(*
SPDX-FileCopyrightText: © 2026 Oleksandr Tiutyk <trofimich@gmail.com>
SPDX-License-Identifier: MIT
License: https://opensource.org/license/mit
*)

(*!
<summary>Selects whether LogManager supplies no number, a global sequence or a sequence per category.</summary>
<description>
Sequences use counters of requests passing filtering, incremented before the logger call. Numbers represent
attempts rather than successful writes; unsuccessful writes can leave gaps in the output sequence.
</description>
*)
{attribute 'qualified_only'}
{attribute 'strict'}
{attribute 'to_string'}
TYPE LOG_MESSAGE_NUMBER_FORMAT :
(
	NONE := 0,
	SEQUENTIAL,
	SEQUENTIAL_BY_CATEGORY
);
END_TYPE

(* stored: Version 1.1.0.1
   DUT LOG_MESSAGE_NUMBER_FORMAT: Id {7db08bfe-99ea-4abc-9ab7-c786550a57d1} *)
